TYPE WcStateBase_A2171C4E :
STRUCT
END_STRUCT
END_TYPE

(* stored: Version 1.2.0.0, ProductVersion 3.1.4024.9
   DUT WcStateBase_A2171C4E: Id {370028f6-e257-4ab8-a232-f9b62cfed262} *)
